(* IEC 61131-3 sources: Caravan/Archiv/12-04-19/Stations/MachineControl/MachineControl/Class/Battery_Class, 1 file *)

(* ---- Battery_Class.st ---- *)
(*!
<Class
	Name               = "Battery_Class"
	Revision           = "0.0"
	RealtimeTask       = "false"
	CyclicTask         = "true"
	DefCyclictime      = "100 ms"
	BackgroundTask     = "false"
	Sigmatek           = "false"
	OSInterface        = "false"
	HighPriority       = "false"
	Automatic          = "false"
	UpdateMode         = "Prescan"
	SharedCommandTable = "true"
	Objectsize         = "(690,300)">
	<Channels>
		<Server Name="ActSystemState" Visualized="true" Initialize="false" WriteProtected="false" Retentive="SRam"/>
		<Server Name="ActualAmps_S" Visualized="true" Initialize="false" WriteProtected="false" Retentive="false"/>
		<Server Name="ActualTowCarAMP_S" Visualized="true" Initialize="false" WriteProtected="false" Retentive="false"/>
		<Server Name="ActualTowCarVoltage_S" Visualized="true" Initialize="false" WriteProtected="false" Retentive="false"/>
		<Server Name="ActualVoltage_S" Visualized="true" Initialize="false" WriteProtected="false" Retentive="false"/>
		<Server Name="AhBalance_S" Visualized="true" Initialize="false" WriteProtected="false" Retentive="SRam"/>
		<Server Name="AhUsedSinceLastFull_S" Visualized="true" Initialize="false" WriteProtected="false" Retentive="SRam"/>
		<Server Name="BattAhRating" Visualized="true" Initialize="false" WriteProtected="false" Retentive="File"/>
		<Server Name="BattFull_S" Visualized="true" Initialize="false" WriteProtected="false" Retentive="File" Comment="Now the battery is green (&gt;75%)&#13;&#10;&#13;&#10;Ladezustand Gelbatt  AGM  Nass&#13;&#10;100 %  12,95 V  &gt; 12,80 V  12,60 V &#13;&#10;75 %  12,74 V  12,55 V  12,36 V &#13;&#10;50 %  12,54 V  12,30 V  12,10 V &#13;&#10;25 %  12,34 V  12,20 V  11,90 V &#13;&#10;0 %  12,10 V  &lt; 12,00 V  11,80 V"/>
		<Server Name="BattLow_S" Visualized="true" Initialize="false" WriteProtected="false" Retentive="File" Comment="At this point the battery is RED (&lt;25%)&#13;&#10;&#13;&#10;Ladezustand Gelbatt  AGM  Nass&#13;&#10;100 %  12,95 V  &gt; 12,80 V  12,60 V &#13;&#10;75 %  12,74 V  12,55 V  12,36 V &#13;&#10;50 %  12,54 V  12,30 V  12,10 V &#13;&#10;25 %  12,34 V  12,20 V  11,90 V &#13;&#10;0 %  12,10 V  &lt; 12,00 V  11,80 V"/>
		<Server Name="BattMax_S" Visualized="true" Initialize="false" WriteProtected="false" Retentive="File" Comment="Max Voltage in mV for battery indicator&#13;&#10;&#13;&#10;&#13;&#10;&#13;&#10;Ladezustand Gelbatt  AGM  Nass&#13;&#10;100 %  12,95 V  &gt; 12,80 V  12,60 V &#13;&#10;75 %  12,74 V  12,55 V  12,36 V &#13;&#10;50 %  12,54 V  12,30 V  12,10 V &#13;&#10;25 %  12,34 V  12,20 V  11,90 V &#13;&#10;0 %  12,10 V  &lt; 12,00 V  11,80 V"/>
		<Server Name="BattMin_S" Visualized="true" Initialize="false" WriteProtected="false" Retentive="File" Comment="Minimal voltage on battery Indicator&#13;&#10;&#13;&#10;Ladezustand Gelbatt  AGM  Nass&#13;&#10;100 %  12,95 V  &gt; 12,80 V  12,60 V &#13;&#10;75 %  12,74 V  12,55 V  12,36 V &#13;&#10;50 %  12,54 V  12,30 V  12,10 V &#13;&#10;25 %  12,34 V  12,20 V  11,90 V &#13;&#10;0 %  12,10 V  &lt; 12,00 V  11,80 V"/>
		<Server Name="ClassSvr" Visualized="false" Initialize="false" WriteProtected="true" Retentive="false"/>
		<Server Name="PercentByVoltage_S" Visualized="true" Initialize="false" WriteProtected="false" Retentive="false"/>
		<Server Name="RemBattAh_S" Visualized="true" Initialize="false" WriteProtected="false" Retentive="SRam"/>
		<Server Name="RESET_AhBalance_S" Visualized="true" Initialize="false" WriteProtected="false" Retentive="false"/>
		<Server Name="RESET_AhUsedSinceLastFull_S" Visualized="true" Initialize="false" WriteProtected="false" Retentive="false"/>
		<Server Name="VoltageOffsetHigh_S" Visualized="true" Initialize="false" WriteProtected="false" Retentive="File"/>
		<Server Name="VoltageOffsetLOW_S" Visualized="true" Initialize="false" WriteProtected="false" Retentive="File"/>
		<Client Name="ActualAmps1_C" Required="true" Internal="false"/>
		<Client Name="ActualAmps2_C" Required="true" Internal="false"/>
		<Client Name="ActualTowCarVoltage_C" Required="true" Internal="false"/>
		<Client Name="ActualVoltage_C" Required="true" Internal="false"/>
	</Channels>
</Class>
*)
Battery_Class : CLASS
  //Servers:
	ClassSvr 	: SvrChCmd_DINT;
	ActSystemState 	: SvrCh_SystemStateType;
	BattMax_S 	: SvrCh_DINT;
	BattMin_S 	: SvrCh_DINT;
	BattLow_S 	: SvrCh_DINT;
	BattFull_S 	: SvrCh_DINT;
	BattAhRating 	: SvrCh_DINT;
	RemBattAh_S 	: SvrCh_DINT;
	ActualVoltage_S 	: SvrCh_DINT;
	VoltageOffsetHigh_S 	: SvrCh_DINT;
	VoltageOffsetLOW_S 	: SvrCh_DINT;
	AhUsedSinceLastFull_S 	: SvrCh_DINT;
	RESET_AhUsedSinceLastFull_S 	: SvrCh_DINT;
	AhBalance_S 	: SvrCh_DINT;
	RESET_AhBalance_S 	: SvrCh_DINT;
	ActualAmps_S 	: SvrCh_DINT;
	ActualTowCarAMP_S 	: SvrCh_DINT;
	ActualTowCarVoltage_S 	: SvrCh_DINT;
	PercentByVoltage_S 	: SvrCh_DINT;
  //Clients:
	ActualAmps1_C 	: CltCh_DINT;
	ActualAmps2_C 	: CltCh_DINT;
	ActualVoltage_C 	: CltCh_DINT;
	ActualTowCarVoltage_C 	: CltCh_DINT;
  //Variables:
		OPS_MerkerVAR 	: UDINT;
		OPS_MerkerVAR2 	: UDINT;
		ReadCounterVAR 	: DINT;
		PrepVar 	: DINT;
		PrepVar2 	: DINT;
		VoltageOffsetVAR 	: DINT;
  //Functions:

	FUNCTION VIRTUAL GLOBAL CyWork
		VAR_INPUT
			EAX 	: UDINT;
		END_VAR
		VAR_OUTPUT
			state (EAX) 	: UDINT;
		END_VAR;
  //Tables:
	FUNCTION @STD
		VAR_OUTPUT
			ret_code	: CONFSTATES;
		END_VAR;
	FUNCTION GLOBAL TAB @CT_;
END_CLASS;

FUNCTION VIRTUAL GLOBAL Battery_Class::CyWork
	VAR_INPUT
		EAX 	: UDINT;
	END_VAR
	VAR_OUTPUT
		state (EAX) 	: UDINT;
	END_VAR

    //Einlesen
    ActualAmps1_C := ActualAmps1_C.Read();

    ActualAmps2_C :=  ActualAmps2_C.Read();

    ActualVoltage_C := ActualVoltage_C.Read();

    ActualTowCarVoltage_C :=  ActualTowCarVoltage_C.Read();

//    case ActSystemState of
//
//
//    	SystemStateType::Charge:
//
//         if ops.tAbsolute - OPS_MerkerVAR2 >= 1000 then
//
//            if  RemBattAh_S <=  (BattAhRating*100) then
//
//                 PrepVar2   :=    RemBattAh_S + (ActualAmps1_C/54);
//
//                 RemBattAh_S  := RemBattAh_S.Write(input:=PrepVar2);
//
//
//                 OPS_MerkerVAR2 :=  ops.tAbsolute;
//
//               ELSE
//
//                PrepVar2  :=  (BattAhRating*100);
//
//                RemBattAh_S :=   RemBattAh_S.Write(input:=PrepVar2);
//
//
//            end_if;
//
//
//
//
//
//         end_if;
//
//
//
//    	  if ActualAmps_S  > 0  then
//
//           if  ActualAmps_S <  500 & ActualVoltage_S > BattFull_S  then
//
//                  AhUsedSinceLastFull_S :=  0;
//
//                  ActSystemState := FullyCarged;
//
//           end_if;
//
//        else
//
//            ActSystemState  :=   Discharge;
//
//        end_if;
//
//
//
//
//
//      SystemStateType::Discharge:
//
//        if ActualAmps_S > 0 then
//
//            ActSystemState  :=  Charge;
//
//        end_if;
//
//
//        if ops.tAbsolute - OPS_MerkerVAR2 >= 1000 then
//
//                 PrepVar2       :=  AhUsedSinceLastFull_S + (ActualAmps1_C/54);//3600 sec, / Mess-shunt Messung :1.5 ergiebt mA * 1000
//
//                 AhUsedSinceLastFull_S.Write(input:=PrepVar2);
//
//
//                 PrepVar2   :=    RemBattAh_S + (ActualAmps1_C/54);
//
//                 RemBattAh_S.Write(input:=PrepVar2);
//
//
//                 OPS_MerkerVAR2 :=  ops.tAbsolute;
//
//         end_if;
//
//
//
//
//      SystemStateType::FullyCarged:
//
//          RemBattAh_S :=  RemBattAh_S.Write(input:=BattAhRating*100);
//
//          AhUsedSinceLastFull_S.Write(input:=0);
//
//
//          if ActualAmps_S > 500 then
//
//                ActSystemState  :=  Charge;
//
//               elsif ActualAmps_S < 0 then
//
//                ActSystemState  :=  Discharge;
//
//          end_if;
//
//
//
//
//
//
//
//    end_case;

//
//    if ops.tAbsolute - OPS_MerkerVAR >= 1000 then
//
//       PrepVar       :=  AhBalance_S + (ActualAmps1_C/54);//3600 sec, / Mess-shunt Messung :1.5 ergiebt mA * 1000
//
//      AhBalance_S.Write(input:=PrepVar);
//
//       OPS_MerkerVAR :=  ops.tAbsolute;
//
//       ReadCounterVAR  +=  1;
//
//    end_if;
//

//Reset AH Balance
//
//    if RESET_AhBalance_S  = true then
//
//        AhBalance_S :=  AhBalance_S.Write(input:=0);
//
//    end_if;

//Reset AH seit letzter Ladung

//    if RESET_AhUsedSinceLastFull_S  = true then
//
//        AhUsedSinceLastFull_S :=  AhUsedSinceLastFull_S.Write(input:=0);
//        ActSystemState        :=  FullyCarged;
//
//    end_if;
//

//    ActualAmps_S    :=    ActualAmps_S.Write(input:=(ActualAmps1_C*10/15));
//
//    ActualTowCarAMP_S :=    ActualTowCarAMP_S.Write(input:=(ActualAmps2_C*10/24)*-1);

    ActualVoltage_S :=    ActualVoltage_S.Write(input:=(ActualVoltage_C * 2));//Spannungsteiler teilt die Spannung daher *2 um zurückturechnen

    ActualTowCarVoltage_S :=    ActualTowCarVoltage_S.Write(input:=(ActualTowCarVoltage_C *2));

    PercentByVoltage_S  :=  (1000000 / BattFull_S) * ActualVoltage_S;

    PercentByVoltage_S  :=  PercentByVoltage_S.Write(input:= PercentByVoltage_S);

	state := READY;

END_FUNCTION
